(**************************************************************************************
 * 	Application		:	BoxControl Framework
 *	Revision		:	$Revision: 404529 $
 *	Revision date	:	$Date: 2018-04-23 08:21:38 +0200 (Mo., 23 Apr 2018) $
 *	Last changed by	:	$Author: b7bolm $
 *	URL				:	$URL: http://almscdc.swisslog.com/repo/SWPD/Development/BoxControlFramework/20_Release/trunk/01_Software/BCF/BCF/JumpStart/20_Product/11_Emu/10_Base/10_Lib/00_GVLs/RegistryEmulation.TcGVL $
 *
 *	Purpose			:	Global registration. All types use the same. (Emulation)
 *
 * ------------------------------------------------------------------------------------
 *	Copyright Swisslog [IP AG], Switzerland. All rights reserved.
 * 
 * ------------------------------------------------------------------------------------
 *	
 * 	Revision History: 
 *
 * 	VERSION			DATE			INITIALS			DESCRIPTION
 *	0.1				01.01.2001		swl					Example
 *
 **************************************************************************************)
VAR_GLOBAL
	FunctionRegistryEmulation	: ARRAY[E_FunctionNumber.F_BEGIN_FUNCTION..E_FunctionNumber.F_END_EXTERN_FUNCTION -1] OF ST_FunctionRegistryConvEmulation; // Function registry
	ElementRegistryEmulation 	: ARRAY[E_ElementNumber.E_BEGIN_ELEMENT..E_ElementNumber.E_END_ELEMENT -1] OF ST_ElementRegistryConvEmulation; // Element registry 
	GroupRegistryEmulation 		: ARRAY[E_GroupNumber.G_BEGIN_GROUP..E_GroupNumber.G_END_GROUP -1] OF ST_GroupRegistryConvEmulation; // Group registry 
	SubsystemRegistryEmulation	: ST_SubsystemRegistryConvEmulation; // Subsystem registry	
END_VAR

(* stored: Version 1.1.0.1, ProductVersion 3.1.4022.12
   GVL RegistryEmulation: Id {1e461a79-92b4-4dab-9bf9-5a19eb626d4c} *)
